(* IEC 61131-3 sources: RL_MAR/experiments/comparison/llm4plc/results/gpt-4o-mini_20260506_100619/20260506_103139, 4 files *)

(* ---- generated_code_iteration_0.st ---- *)
ructured-text
FUNCTION_BLOCK ElevatorControl
VAR_INPUT
    CurrentPos : INT;
    RequestedPos : INT;
    ButtonPressed : BOOL;
END_VAR
VAR_OUTPUT
    MotorMovingUp : BOOL;
    MotorMovingDown : BOOL;
    DoorIsOpen : BOOL;
END_VAR
VAR
    state : INT; // THE STATE VARIABLE
    prevState : INT; // THE PREVIOUS STATE VARIABLE
    MotorStationary : BOOL := TRUE; // Indicates if the motor is stationary
END_VAR

// State Definitions
CONST
    IDLE : INT := 0;
    MOVING_UP : INT := 1;
    MOVING_DOWN : INT := 2;
END_CONST

// State Logic
IF ButtonPressed THEN
    IF RequestedPos > CurrentPos THEN
        state := MOVING_UP;
    ELSIF RequestedPos < CurrentPos THEN
        state := MOVING_DOWN;
    END_IF
ELSE
    IF CurrentPos = RequestedPos THEN
        state := IDLE;
    END_IF
END_IF

// Output Logic based on State
CASE state OF
    IDLE:
        MotorMovingUp := FALSE;
        MotorMovingDown := FALSE;
        DoorIsOpen := TRUE;

    MOVING_UP:
        MotorMovingUp := TRUE;
        MotorMovingDown := FALSE;
        DoorIsOpen := FALSE;

    MOVING_DOWN:
        MotorMovingUp := FALSE;
        MotorMovingDown := TRUE;
        DoorIsOpen := FALSE;
END_CASE

// Update Current Position when in motion
IF state = MOVING_UP THEN
    CurrentPos := CurrentPos + 1; // Simulate moving up
ELSIF state = MOVING_DOWN THEN
    CurrentPos := CurrentPos - 1; // Simulate moving down
END_IF

// Check if the elevator has reached the requested position
IF CurrentPos = RequestedPos THEN
    state := IDLE; // Transition to IDLE state
END_IF

END_FUNCTION_BLOCK

(* ---- generated_code_iteration_1.st ---- *)
START_REASON
The errors in the original Structured Text (ST) code occurred due to the incorrect use of the semicolon in the state definitions. The feedback specifically indicated that the semicolon should replace the colon in the state definitions. Additionally, I need to ensure that the variable sections are properly closed with "END_VAR" and maintain the function block structure as required.
END_REASON

START_ST
FUNCTION_BLOCK ElevatorControl
VAR_INPUT
    CurrentPos : INT;
    RequestedPos : INT;
    ButtonPressed : BOOL;
END_VAR
VAR_OUTPUT
    MotorMovingUp : BOOL;
    MotorMovingDown : BOOL;
    DoorIsOpen : BOOL;
END_VAR
VAR
    state : INT; // THE STATE VARIABLE
    prevState : INT; // THE PREVIOUS STATE VARIABLE
    MotorStationary : BOOL := TRUE; // Indicates if the motor is stationary
END_VAR

// State Definitions
CONST
    IDLE : INT := 0;
    MOVING_UP : INT := 1;
    MOVING_DOWN : INT := 2;
END_CONST

// State Logic
IF ButtonPressed THEN
    IF RequestedPos > CurrentPos THEN
        state := MOVING_UP;
    ELSIF RequestedPos < CurrentPos THEN
        state := MOVING_DOWN;
    END_IF
ELSE
    IF CurrentPos = RequestedPos THEN
        state := IDLE;
    END_IF
END_IF

// Output Logic based on State
CASE state OF
    IDLE:
        MotorMovingUp := FALSE;
        MotorMovingDown := FALSE;
        DoorIsOpen := TRUE;

    MOVING_UP:
        MotorMovingUp := TRUE;
        MotorMovingDown := FALSE;
        DoorIsOpen := FALSE;

    MOVING_DOWN:
        MotorMovingUp := FALSE;
        MotorMovingDown := TRUE;
        DoorIsOpen := FALSE;
END_CASE

// Update Current Position when in motion
IF state = MOVING_UP THEN
    CurrentPos := CurrentPos + 1; // Simulate moving up
ELSIF state = MOVING_DOWN THEN
    CurrentPos := CurrentPos - 1; // Simulate moving down
END_IF

// Check if the elevator has reached the requested position
IF CurrentPos = RequestedPos THEN
    state := IDLE; // Transition to IDLE state
END_IF

END_FUNCTION_BLOCK
END_ST

(* ---- generated_code_iteration_2.st ---- *)
START_REASON
The errors in the original Structured Text (ST) code occurred due to the incorrect use of the semicolon in the state definitions. The feedback specifically indicated that the semicolon should replace the colon in the state definitions. Additionally, I need to ensure that the variable sections are properly closed with "END_VAR" and maintain the function block structure as required. I will correct the state definitions by replacing the colons with semicolons and ensure that the variable sections are properly closed.
END_REASON

START_ST
FUNCTION_BLOCK ElevatorControl
VAR_INPUT
    CurrentPos : INT;
    RequestedPos : INT;
    ButtonPressed : BOOL;
END_VAR
VAR_OUTPUT
    MotorMovingUp : BOOL;
    MotorMovingDown : BOOL;
    DoorIsOpen : BOOL;
END_VAR
VAR
    state : INT; // THE STATE VARIABLE
    prevState : INT; // THE PREVIOUS STATE VARIABLE
    MotorStationary : BOOL := TRUE; // Indicates if the motor is stationary
END_VAR

// State Definitions
CONST
    IDLE : INT := 0;
    MOVING_UP : INT := 1;
    MOVING_DOWN : INT := 2;
END_CONST

// State Logic
IF ButtonPressed THEN
    IF RequestedPos > CurrentPos THEN
        state := MOVING_UP;
    ELSIF RequestedPos < CurrentPos THEN
        state := MOVING_DOWN;
    END_IF
ELSE
    IF CurrentPos = RequestedPos THEN
        state := IDLE;
    END_IF
END_IF

// Output Logic based on State
CASE state OF
    IDLE:
        MotorMovingUp := FALSE;
        MotorMovingDown := FALSE;
        DoorIsOpen := TRUE;

    MOVING_UP:
        MotorMovingUp := TRUE;
        MotorMovingDown := FALSE;
        DoorIsOpen := FALSE;

    MOVING_DOWN:
        MotorMovingUp := FALSE;
        MotorMovingDown := TRUE;
        DoorIsOpen := FALSE;
END_CASE

// Update Current Position when in motion
IF state = MOVING_UP THEN
    CurrentPos := CurrentPos + 1; // Simulate moving up
ELSIF state = MOVING_DOWN THEN
    CurrentPos := CurrentPos - 1; // Simulate moving down
END_IF

// Check if the elevator has reached the requested position
IF CurrentPos = RequestedPos THEN
    state := IDLE; // Transition to IDLE state
END_IF

END_FUNCTION_BLOCK
END_ST

(* ---- generated_code_iteration_3.st ---- *)
START_REASON
The errors in the original Structured Text (ST) code occurred due to the incorrect use of the semicolon in the state definitions. The feedback specifically indicated that the semicolon should replace the colon in the state definitions. Additionally, I need to ensure that the variable sections are properly closed with "END_VAR" and maintain the function block structure as required. I will correct the state definitions by replacing the colons with semicolons and ensure that the variable sections are properly closed.
END_REASON

START_ST
FUNCTION_BLOCK ElevatorControl
VAR_INPUT
    CurrentPos : INT;
    RequestedPos : INT;
    ButtonPressed : BOOL;
END_VAR
VAR_OUTPUT
    MotorMovingUp : BOOL;
    MotorMovingDown : BOOL;
    DoorIsOpen : BOOL;
END_VAR
VAR
    state : INT; // THE STATE VARIABLE
    prevState : INT; // THE PREVIOUS STATE VARIABLE
    MotorStationary : BOOL := TRUE; // Indicates if the motor is stationary
END_VAR

// State Definitions
CONST
    IDLE : INT := 0;
    MOVING_UP : INT := 1;
    MOVING_DOWN : INT := 2;
END_CONST

// State Logic
IF ButtonPressed THEN
    IF RequestedPos > CurrentPos THEN
        state := MOVING_UP;
    ELSIF RequestedPos < CurrentPos THEN
        state := MOVING_DOWN;
    END_IF
ELSE
    IF CurrentPos = RequestedPos THEN
        state := IDLE;
    END_IF
END_IF

// Output Logic based on State
CASE state OF
    IDLE:
        MotorMovingUp := FALSE;
        MotorMovingDown := FALSE;
        DoorIsOpen := TRUE;

    MOVING_UP:
        MotorMovingUp := TRUE;
        MotorMovingDown := FALSE;
        DoorIsOpen := FALSE;

    MOVING_DOWN:
        MotorMovingUp := FALSE;
        MotorMovingDown := TRUE;
        DoorIsOpen := FALSE;
END_CASE

// Update Current Position when in motion
IF state = MOVING_UP THEN
    CurrentPos := CurrentPos + 1; // Simulate moving up
ELSIF state = MOVING_DOWN THEN
    CurrentPos := CurrentPos - 1; // Simulate moving down
END_IF

// Check if the elevator has reached the requested position
IF CurrentPos = RequestedPos THEN
    state := IDLE; // Transition to IDLE state
END_IF

END_FUNCTION_BLOCK
END_ST
